// TIA Portal V19 export
ORGANIZATION_BLOCK "Main"   // OB2401, LAD, ProgramCycle
TITLE = "Main Program Sweep (Cycle)"
// stored: AutoNumber false, Namespace Unit2.EM3, SetENOAutomatically false
   VAR_INPUT
      Initial_Call : Bool;   // Initial call of this OB
      Remanence : Bool;   // =True, if remanent data are available
   END_VAR
BEGIN

REGION Network 1
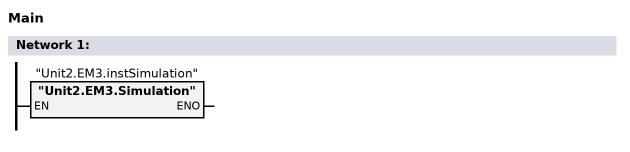
   RUNG wire#powerrail
      "Unit2.EM3.instSimulation"()
   END_RUNG
   // the same network as SCL:
   "Unit2.EM3.instSimulation"();   // "Unit2.EM3.Simulation"
END_REGION

REGION Network 2 (SCL)
   "Unit2.EM3.CallEquipment_DB"(unitStatus:="Unit2.EmNodes".unitStatus,
                    unitAlarmDB:="Unit2.Alarms".emAlarms[Unit2_EM3],
                    emFeedback:="Unit2.EmNodes".emFeedback[Unit2_EM3]);
END_REGION
END_ORGANIZATION_BLOCK
